(* PLC project PLC, Beckhoff Automation GmbH TwinCAT PLC Control 3.5.13.21 *)
(* stored: creationDateTime 2024-02-17T22:42:49.4999772, modificationDateTime 2024-02-17T22:42:49.4999772 *)

TYPE CylInput :
STRUCT
	posFw AT %I*: BOOL;
	posRv AT %I*: BOOL;
END_STRUCT
END_TYPE
